(* CoDeSys 2.3 export: WRITEBIT.EXP *)

(* POU Functions/WriteBit, ST *)
FUNCTION WriteBit : BOOL
VAR_INPUT
	pBit : POINTER TO BOOL ; (**< AddressValue of the target *)
	bValue : BOOL ; (**< Value to equalize bit to *)
END_VAR
VAR
END_VAR
pBit^ := bValue;
END_FUNCTION
